// TwinCAT 3 PLC project PLC_ST03
// ProgramVersion: 3.1.4024.0
// libraries:
//   Base Objects Library, * (JABIL RAC LATAM)
//   Tc2_MC2, * (Beckhoff Automation GmbH)
//   Tc2_Standard, * (Beckhoff Automation GmbH)
//   Tc2_System, * (Beckhoff Automation GmbH)
//   Tc3_Module, * (Beckhoff Automation GmbH)
// project tree:
//   / PlcST03Task.TcTTO
//   POUs/00-Main/ MAIN_ST03.TcPOU
// (motion and I/O tree: see PLC project plc_st01)
// real-time tasks:
//   TASK PlcST01Task: cycle T#10ms, priority 20, ADS port 350
//   TASK PlcST02Task: cycle T#10ms, priority 21, ADS port 351
//   TASK PlcST03Task: cycle T#10ms, priority 22, ADS port 352
// variable links:

CONFIGURATION PLC_ST03
    RESOURCE PLC ON TwinCAT3
        TASK PlcST03Task(INTERVAL := T#10ms, PRIORITY := 22);
        PROGRAM MAIN_ST03 WITH PlcST03Task : MAIN_ST03;
    END_RESOURCE
END_CONFIGURATION

// ---- POUs/00-Main/MAIN_ST03.TcPOU
PROGRAM MAIN_ST03
VAR
	fbStation03							: RACBaseObjects.FB_Station;
END_VAR

fbStation03(bInitFinished := FALSE);

END_PROGRAM
